FUNCTION_BLOCK FB_StirringModule
VAR_INPUT
END_VAR
VAR_OUTPUT
END_VAR
VAR
END_VAR

END_FUNCTION_BLOCK

(* stored: Version 1.1.0.1
   POU FB_StirringModule: Id {56fbbf30-5d64-4ae6-8093-f8ba13294201}, SpecialFunc None *)
